Staubli VAL3: OnF4.pgx

program OnF4()
begin
  call Pallet:start()
  bUserRefresh=true
end
